# EPICS autosave request: vici/sixteenGasSelect_2EMT_1VALVE_positions.req
$(P)$(Q):SELECT.EIST
$(P)$(Q):SELECT.ELST
$(P)$(Q):SELECT.FFST
$(P)$(Q):SELECT.FRST
$(P)$(Q):SELECT.FTST
$(P)$(Q):SELECT.FVST
$(P)$(Q):SELECT.NIST
$(P)$(Q):SELECT.ONST
$(P)$(Q):SELECT.SVST
$(P)$(Q):SELECT.SXST
$(P)$(Q):SELECT.TEST
$(P)$(Q):SELECT.THST
$(P)$(Q):SELECT.TTST
$(P)$(Q):SELECT.TVST
$(P)$(Q):SELECT.TWST
$(P)$(Q):SELECT.ZRST
$(P)$(Q):STR1
$(P)$(Q):STR2
$(P)$(Q):STR3
$(P)$(Q):STR4
